{attribute 'qualified_only'}
{attribute 'strict'}
TYPE E_SMPTE_PartOfFrame :
(
	first := 0, second := 1
)BYTE;
END_TYPE

(* stored: Version 1.1.0.1, ProductVersion 3.1.4024.12
   DUT E_SMPTE_PartOfFrame: Id {b56707d9-2934-4a2c-8486-7fcadb2d9724} *)
